{attribute 'linkalways'} 
{attribute 'no_explicit_call' := 'This FB is a CLASS and must be accessed using methods or properties'}
{attribute 'enable_dynamic_creation'}
FUNCTION_BLOCK WriteBoolToBitOperation EXTENDS Disposable IMPLEMENTS I_DatatypeOperation
VAR
	source : REFERENCE TO _BOOL;
	destination : I_BIT;
END_VAR

METHOD Execute
VAR
END_VAR
destination.Value := source.Value;
END_METHOD

METHOD FB_init : BOOL
VAR_INPUT
	bInitRetains : BOOL; // if TRUE, the retain variables are initialized (warm start / cold start)
	bInCopyCode : BOOL;  // if TRUE, the instance afterwards gets moved into the copy code (online change)
	Source : REFERENCE TO _BOOL;
	Destination : I_BIT;
END_VAR
THIS^.source REF= Source;
THIS^.destination := Destination;
END_METHOD

END_FUNCTION_BLOCK

(* stored: Version 1.1.0.1, ProductVersion 3.1.4024.15
   POU WriteBoolToBitOperation: Id {77960676-50e4-46ca-9a25-2dc838a8dff5}, SpecialFunc None
   Folder Constructor: Id {b9064319-43a5-47f9-834f-c427a5e1a32f}
   Method Execute: Id {0eb96d2c-ecad-4b74-b2fa-67b43b1b6d7d}
   Method FB_init: Id {0d2c3979-8f8c-4763-947a-548c8c43a736} *)
